PROGRAM MAIN
VAR
	diKapSensor1 AT %I* : BOOL ;
	bMinneKapSensor1 : BOOL := 0;
	diKapSensor2 AT %I* : BOOL ;
	bMinneKapSensor2 : BOOL := 0;
	bMinneKap_OR : BOOL := 0;
	bMinneKap_AND : BOOL := 0;
END_VAR

bMinneKapSensor1 := diKapSensor1 ;
bMinneKapSensor2 := diKapSensor2 ;
bMinneKap_OR := diKapSensor1 OR diKapSensor2 ;
bMinneKap_AND := diKapSensor1 AND diKapSensor2 ;

END_PROGRAM

(* stored: Version 1.1.0.1, ProductVersion 3.1.4024.9
   POU MAIN: Id {b33fd355-6fbe-4b45-9d16-bcb82b21ff75}, SpecialFunc None *)
